// TIA Portal V20 export
TYPE "s_PLC_Interlocks"
// stored: Access Published, IsFailsafeCompliant true, Namespace Safety
   STRUCT
      "Connection status" { ExternalWritable := 'False'; S7_SetPoint := 'True'} : "Safety.s_CONNECTION_STATUS";
      CellInterlocks { ExternalWritable := 'False'; S7_SetPoint := 'True'} : "Safety.s_zc_CellInterlocks";
      InterlockToAdjCellICSD { ExternalWritable := 'False'; S7_SetPoint := 'True'} : "Safety.s_zc_IntercellSafetyDeviceToAdjCell";
      NormalInterlocks { S7_SetPoint := 'True'} : "Safety.s_zc_NormalInterlocks";
      MiscInterlock { S7_SetPoint := 'True'} : "Safety.s_zc_MiscInterlocks";
   END_STRUCT;
   // // NormalInterlocks.reserved02 : BA60 JR PP Left Door Normal Open (Stacker#1)
   // // NormalInterlocks.reserved03 : BA60 Top Tape Door Normal Open (Stacker#2)
   // // NormalInterlocks.reserved04 : BA60 JR PP Left Door Forced Open (Stacker#1)
   // // NormalInterlocks.reserved05 : BA60 Top Tape Door Forced Open (Stacker#2)
   // // NormalInterlocks.reserved06 : BA60 External Door Open (Stacker#1)
   // // NormalInterlocks.reserved07 : BA60 External Door Open (Stacker#2)
   // // NormalInterlocks.reserved08 : Cathode Conveyor Cover Closed
   // // NormalInterlocks.reserved09 : Anode Conveyor Cover Closed
   // // NormalInterlocks.reserved10 : BA60 Light Curtain Muting (Stacker#1)
   // // NormalInterlocks.reserved11 : BA60 Light Curtain NOK (Stacker#1)
   // // NormalInterlocks.reserved12 : BA60 Light Curtain Muting (Stacker#2)
   // // NormalInterlocks.reserved13 : BA60 Light Curtain NOK (Stacker#2)
END_TYPE
